Fanuc TP program (LS listing): wrong_order.ls

/ATTR
OWNER		= MNEDITOR;
COMMENT		= "";
PROG_SIZE	= 100;
CREATE		= DATE 25-01-01  TIME 00:00:00;
MODIFIED	= DATE 25-01-01  TIME 00:00:00;
FILE_NAME	= ;
VERSION		= 0;
LINE_COUNT	= 1;
MEMORY_SIZE	= 100;
PROTECT		= READ_WRITE;
TCD:  STACK_SIZE	= 0,
      TASK_PRIORITY	= 50,
      TIME_SLICE	= 0,
      BUSY_LAMP_OFF	= 0,
      ABORT_REQUEST	= 0,
      PAUSE_REQUEST	= 0;
DEFAULT_GROUP	= 1,*,*,*,*;
CONTROL_CODE	= 00000000 00000000;
/PROG  WRONGORD
/APPL
/MN
   1:   ;
/POS
/END
